// Mitsubishi GX Works2 project: 230927-001-hello word   PLC: Q03UDV

// task Task_01 (event TRUE, interval 0, priority 31): POU_01

PROGRAM POU_01
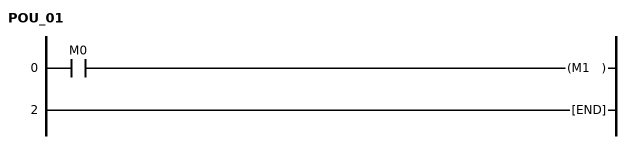
0     LD      M0
      OUT     M1
2     END
END_PROGRAM
